FUNCTION_BLOCK OBJ_Carrier IMPLEMENTS I_Carrier
VAR_INPUT
END_VAR
VAR_OUTPUT
END_VAR
VAR
	//--s_eLocation : E_Location;
	//--s_eLocationPrev : E_Location;
	//--s_eDestination : E_Location;
	
	//--s_bCheckedAtInfeed : BOOL;
	//--s_bAlligned : BOOL;
	//--s_bDocked : BOOL;
	//--s_bUnDocked : BOOL;
	//--s_bFlushed : BOOL;
	
	
	
END_VAR

METHOD PUBLIC m_initNewCarrier : BOOL
VAR_INPUT
	i_eDestination : E_Location := E_Location.UNKNOWN;
END_VAR

s_eLocation := E_Location.INFEED;
s_eLocationPrev := E_Location.INFEED;
s_eDestination := i_eDestination;
	
s_bCheckedAtInfeed := FALSE;
s_bAlligned := FALSE;
s_bDocked := FALSE;
s_bUnDocked := FALSE;
s_bFlushed := FALSE;
END_METHOD

PROPERTY PUBLIC p_bAlligned : BOOL
GET
END_GET
SET
END_SET
END_PROPERTY

PROPERTY PUBLIC p_bFlushedClean : BOOL
GET
END_GET
SET
END_SET
END_PROPERTY

PROPERTY PUBLIC p_eDestination : E_Location
GET
END_GET
SET
END_SET
END_PROPERTY

PROPERTY PUBLIC p_eLocation : E_Location
GET
END_GET
SET
END_SET
END_PROPERTY

PROPERTY PUBLIC p_eLocationPrev : E_Location
GET
END_GET
SET
END_SET
END_PROPERTY

END_FUNCTION_BLOCK

(* stored: Version 1.1.0.1, ProductVersion 3.1.4024.12
   POU OBJ_Carrier: Id {788a2610-a427-4d98-80b8-1d15416d7282}, SpecialFunc None
   Method m_initNewCarrier: Id {234cad66-503e-431c-8f10-335fb71fd3a2}
   Property p_bAlligned: Id {d69c5412-5c2c-45b4-8be3-5444487f9c4a}
   Get Get: Id {91ff997c-7b50-43ae-8859-6bc029d4a907}
   Set Set: Id {1b159a04-f5d9-40fc-a788-b805f96673f4}
   Property p_bFlushedClean: Id {f3ffe3a1-4925-48a7-a230-3a8593a53515}
   Get Get: Id {c309fdb1-b242-4932-9a08-2959c4f7d4a0}
   Set Set: Id {c44cc6d5-fbb2-491f-9876-6b9fc7b7d2e7}
   Property p_eDestination: Id {b5c2a005-f24c-47c7-b596-cc92f8422147}
   Get Get: Id {075c546d-dc3e-46d0-805f-bdc70e2e2a56}
   Set Set: Id {6cd2da6a-84f6-4ca1-8c2b-5f4f7367fdf3}
   Property p_eLocation: Id {a5592312-8b05-45c5-a594-5a434b6a0aac}
   Get Get: Id {242ea7ea-80d9-4806-8bd8-b9f5478cdc71}
   Set Set: Id {6a798601-b837-4016-ace2-8fef13d6ed07}
   Property p_eLocationPrev: Id {429995c5-dd26-4805-b511-29aa571c98b5}
   Get Get: Id {13184503-88fb-4097-accb-94e98c6eefde}
   Set Set: Id {9fb3e566-850e-45bf-928c-e9f879f9415f} *)
